FUNCTION_BLOCK ytimer2
  (* Standard: 61499-2 *)
  (* Version 0.1, 2015-00-20, Th?o, PC_THEO *)
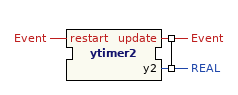
  EVENT_INPUT
    restart;
  END_EVENT
  EVENT_OUTPUT
    update WITH y2;
  END_EVENT
  VAR_OUTPUT
    y2 : REAL;
  END_VAR
  VAR
    d : REAL;
  END_VAR
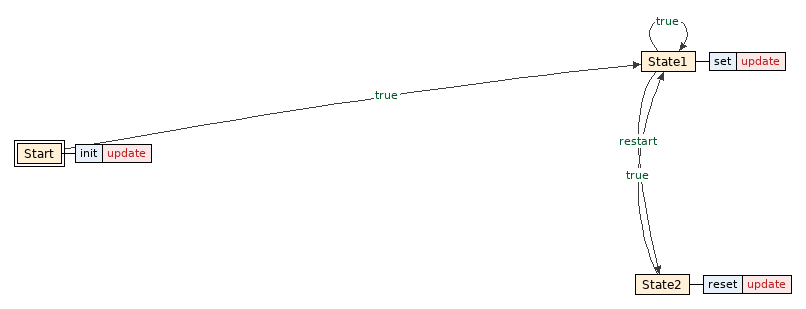
  EC_STATES
    Start : init -> update;
    State1 : set -> update;
    State2 : reset -> update;
  END_STATES
  EC_TRANSITIONS
    Start TO State1 := true;
    State1 TO State2 := restart;
    State1 TO State1 := true;
    State2 TO State1 := true;
  END_TRANSITIONS
  ALGORITHM init IN C:
me->y2=20;
me->d=0.01;
  END_ALGORITHM
  ALGORITHM set IN C:
me->y2=me->y2+me->d;
  END_ALGORITHM
  ALGORITHM reset IN C:
me->y2=0;
  END_ALGORITHM
END_FUNCTION_BLOCK
